// TIA Portal V15.1 export
// export: Created 2024-06-21T08:41:01.898082Z, ExportSetting WithDefaults, DisplayName Totally Integrated Automation Portal, DisplayVersion V15.1 Update 5, DisplayName TIA Portal Openness, DisplayVersion V15.1 Update 5, DisplayName SINAMICS Startdrive Advanced, DisplayVersion V15.1, DisplayName G130, G150, S120, S150, SINAMICS MV, S210, DisplayVersion V15.1, DisplayName G110M, G120, G120C, G120D, G120P, DisplayVersion V15.1, DisplayName STEP 7 Professional, DisplayVersion V15.1 Update 5, DisplayName STEP 7 Safety, DisplayVersion V15.1, DisplayName WinCC Professional, DisplayVersion V15.1 Update 5, DisplayName SIMATIC Visualization Architect, DisplayVersion V15.1
FUNCTION_BLOCK "LMovFnc2Pos"   // FB1102, FBD
TITLE = LMovFnc2Pos
{ S7_Optimized_Access := 'TRUE' }
AUTHOR : VCC
FAMILY : Tooling
VERSION : 0.1
// =============================================================================
// This module will be used for the steering of a two Position movement.
// It will get the commands from different Modes, evaluate the status of the 
// Interlock and give the command to the Actuator or direct to simple outputs.
// =============================================================================
// stored: AutoNumber false, IsIECCheckEnabled false, IsRetainMemResEnabled false, MemoryReserve 100, SetENOAutomatically False, UDAEnableTagReadback false
   VAR_INPUT
      I_PosSet { ExternalAccessible := 'False'; ExternalVisible := 'False'; ExternalWritable := 'False'} : Bool;   // Position Set detection or summary / Position Set Detection
      I_PosRes { ExternalAccessible := 'False'; ExternalVisible := 'False'; ExternalWritable := 'False'} : Bool;   // Position Reset detection or summary / Position Reset Detection
      I_PBSet { ExternalAccessible := 'False'; ExternalVisible := 'False'; ExternalWritable := 'False'} : Bool;   // Push button for Set direction (used in manual with button OP panels )
      I_PBReset { ExternalAccessible := 'False'; ExternalVisible := 'False'; ExternalWritable := 'False'} : Bool;   // Push button for reset direcion (used in manual with pushbutton OP panels) / Push button for Reset direction (used in manual with Pushbutton OP panels)
      I_SetBegin { ExternalAccessible := 'False'; ExternalVisible := 'False'; ExternalWritable := 'False'} : Bool;   // Function Set begin selection
      I_ResBegin { ExternalAccessible := 'False'; ExternalVisible := 'False'; ExternalWritable := 'False'} : Bool;   // Function Reset begin selection
      I_SetIntlkOK { ExternalAccessible := 'False'; ExternalVisible := 'False'; ExternalWritable := 'False'} : Bool;   // Set Interlock
      I_ResIntlkOK { ExternalAccessible := 'False'; ExternalVisible := 'False'; ExternalWritable := 'False'} : Bool;   // Reset Interlock
      I_SafetyOk { ExternalAccessible := 'False'; ExternalVisible := 'False'; ExternalWritable := 'False'} : Bool;   // Safety Ok
      I_HardwareOk { ExternalAccessible := 'False'; ExternalVisible := 'False'; ExternalWritable := 'False'} : Bool;   // Safety Ok / Hardware Ok
   END_VAR
   VAR_OUTPUT
      O_CmdSet { ExternalAccessible := 'False'; ExternalVisible := 'False'; ExternalWritable := 'False'} : Bool;   // Command to activate Set movement / Command to Activate Set movement
      O_CmdRes { ExternalAccessible := 'False'; ExternalVisible := 'False'; ExternalWritable := 'False'} : Bool;   // Command to activate Reset movement / Command to Activate Reset movement
      O_FuncRunning { ExternalAccessible := 'False'; ExternalVisible := 'False'; ExternalWritable := 'False'} : Bool;   // Signal that the function is running
      O_FuncBusyTM { ExternalAccessible := 'False'; ExternalVisible := 'False'; ExternalWritable := 'False'} : Bool;   // Memory Signal that the function is busy
      O_SetFinished { ExternalAccessible := 'False'; ExternalVisible := 'False'; ExternalWritable := 'False'} : Bool;   // Function Set finished to Master Sequencing
      O_ResFinished { ExternalAccessible := 'False'; ExternalVisible := 'False'; ExternalWritable := 'False'} : Bool;   // Function Reset finished to Master Sequencing
      O_IntlkSetAlm { ExternalAccessible := 'False'; ExternalVisible := 'False'; ExternalWritable := 'False'} : Bool;   // Alarm interlock Set / Alarm Interlock Set
      O_IntlkResAlm { ExternalAccessible := 'False'; ExternalVisible := 'False'; ExternalWritable := 'False'} : Bool;   // Alarm interlock Reset / Alarm Interlock Reset
      O_FuncIsSelInMan { ExternalAccessible := 'False'; ExternalVisible := 'False'; ExternalWritable := 'False'} : Bool;   // The function is selected in manual mode / The function is Selected in manual Mode
      O_LED { ExternalAccessible := 'False'; ExternalVisible := 'False'; ExternalWritable := 'False'} : Bool;   // LED-indication / LED - Indication
      O_AlarmABCondition { ExternalAccessible := 'False'; ExternalVisible := 'False'; ExternalWritable := 'False'} : Bool;   // Alarms AB condition / Alarm AB Condition
   END_VAR
   VAR_IN_OUT
      IO_Modes : "Modes";   // Modes
      H_HMI : "H_HMI";   // Animation
      H_MovFnc2Pos : "H_MovFnc2Pos";   // Animation
      H_FncSelInHMI { ExternalAccessible := 'False'; ExternalVisible := 'False'; ExternalWritable := 'False'} : Bool;   // This function is selected to run from HMI / This function is Selected to run from HMI
      C_AlarmResetUsed { ExternalAccessible := 'False'; ExternalVisible := 'False'; ExternalWritable := 'False'} : Bool;   // If true, the alrms will be stored untill reseted / If TRUE The Alarms will be stored untill Reseted
      C_EnableMemBegin { ExternalAccessible := 'False'; ExternalVisible := 'False'; ExternalWritable := 'False'} : Bool;   // Enable memory Begin (Command request is memorised until pos reached) / Enable memory Begin (Command Request is memorised until pos reached)
      C_EnIntlkAlm { ExternalAccessible := 'False'; ExternalVisible := 'False'; ExternalWritable := 'False'} : Bool := TRUE;   // Enable Interlock Alarm
      C_SetReset { ExternalAccessible := 'False'; ExternalVisible := 'False'; ExternalWritable := 'False'} : Bool;   // Enable Set Reset Functionality ( If enabled output is kept until the Cmd direction is changed )
      C_ManualClampCmdSet { ExternalAccessible := 'False'; ExternalVisible := 'False'; ExternalWritable := 'False'} : Bool;   // Manual Clamp Set
      C_ManualClampCmdRes { ExternalAccessible := 'False'; ExternalVisible := 'False'; ExternalWritable := 'False'} : Bool;   // Manual Clamp Reset
      C_ForceManual { ExternalAccessible := 'False'; ExternalVisible := 'False'; ExternalWritable := 'False'} : Bool := FALSE;   // Force Manual
   END_VAR
   VAR
      ResetAlarm { ExternalAccessible := 'False'; ExternalVisible := 'False'; ExternalWritable := 'False'} : Bool;   // Reset Alarm Memory
      CmdSetRequest { ExternalAccessible := 'False'; ExternalVisible := 'False'; ExternalWritable := 'False'} : Bool;   // Set Command request to activate the interlock / Set Command Request to Activate the Interlock
      CmdResRequest { ExternalAccessible := 'False'; ExternalVisible := 'False'; ExternalWritable := 'False'} : Bool;   // Reset Command request to activate the interlock / Reset Command Request to Activate the Interlock
      EdgeStopDetSet { ExternalAccessible := 'False'; ExternalVisible := 'False'; ExternalWritable := 'False'} : Bool;   // Edge on stop detection to be abble to go over it in force manual
      EdgeStopDetRes { ExternalAccessible := 'False'; ExternalVisible := 'False'; ExternalWritable := 'False'} : Bool;   // Edge on stop detection to be abble to go over it in force manual
      IntlkSetAlm { ExternalAccessible := 'False'; ExternalVisible := 'False'; ExternalWritable := 'False'} : Bool;   // Alarm interlock Set / Alarm Interlock Set
      IntlkResAlm { ExternalAccessible := 'False'; ExternalVisible := 'False'; ExternalWritable := 'False'} : Bool;   // Alarm interlock Reset / Alarm Interlock Reset
      CmdSet { ExternalAccessible := 'False'; ExternalVisible := 'False'; ExternalWritable := 'False'} : Bool;   // Command to activate Set movement / Command to Activate Set movement
      CmdRes { ExternalAccessible := 'False'; ExternalVisible := 'False'; ExternalWritable := 'False'} : Bool;   // Command to activate Reset movement / Command to Activate Reset movement
      IntlkSetAlmCond { ExternalAccessible := 'False'; ExternalVisible := 'False'; ExternalWritable := 'False'} : Bool;   // Alarm interlock Set condition / Alarm Interlock Set condition
      IntlkResAlmCond { ExternalAccessible := 'False'; ExternalVisible := 'False'; ExternalWritable := 'False'} : Bool;   // Alarm interlock Reset condition / Alarm Interlock Reset condition
      FuncRunning { ExternalAccessible := 'False'; ExternalVisible := 'False'; ExternalWritable := 'False'} : Bool;   // Function is running
      FuncBusyTM { ExternalAccessible := 'False'; ExternalVisible := 'False'; ExternalWritable := 'False'} : Bool;   // Memory Signal that the function is busy
      AlmFilterResult { ExternalAccessible := 'False'; ExternalVisible := 'False'; ExternalWritable := 'False'} : Bool;   // Alarm filter result
      _AlarmTimer { ExternalAccessible := 'False'; ExternalVisible := 'False'; ExternalWritable := 'False'} : "LTimer";
   END_VAR
   VAR_TEMP   // added for the SCL form of the ladder/FBD networks
      _w1 : Bool;
   END_VAR
BEGIN

REGION Network 1: **** 2.2 - Alarms - Alarm Generation **** Alarm Filter
   // Alarm Filter
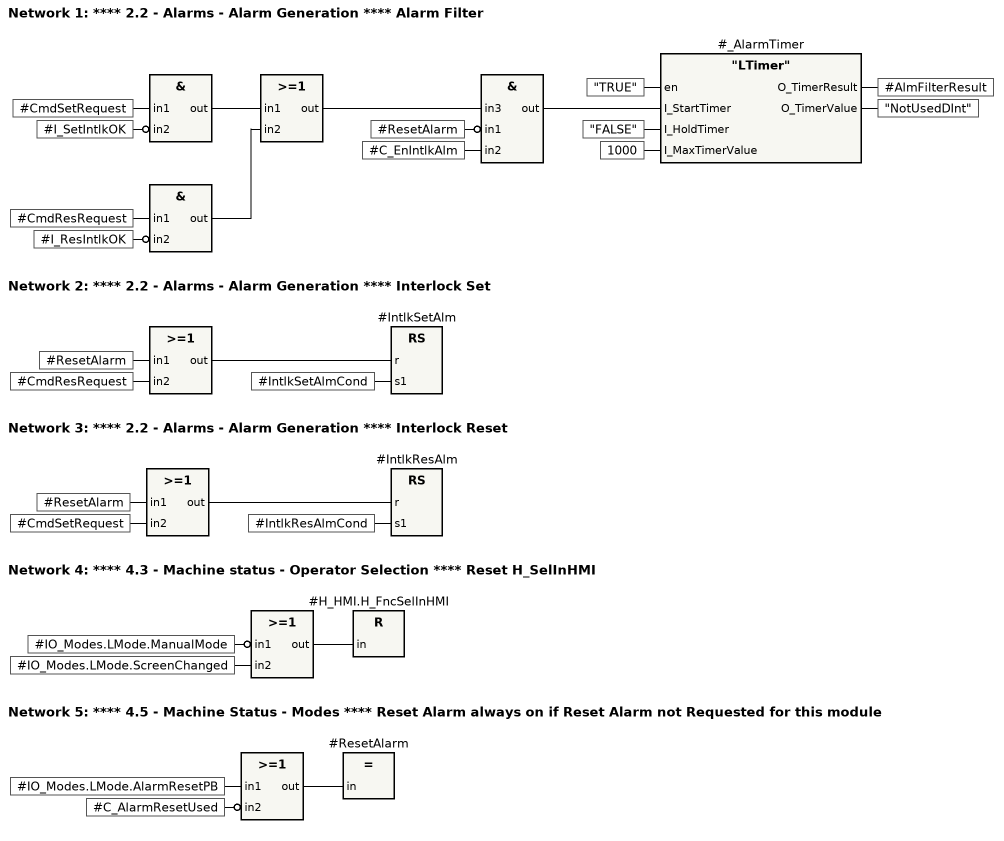
   IF "TRUE" THEN
       #_AlarmTimer(I_StartTimer := ((#CmdSetRequest AND NOT #I_SetIntlkOK) OR (#CmdResRequest AND NOT #I_ResIntlkOK)) AND NOT #ResetAlarm AND #C_EnIntlkAlm,   // "LTimer"
                    I_HoldTimer := "FALSE",
                    I_MaxTimerValue := 1000,
                    O_TimerResult => #AlmFilterResult,
                    O_TimerValue => "NotUsedDInt");
   END_IF;
END_REGION

REGION Network 2: **** 2.2 - Alarms - Alarm Generation **** Interlock Set
   // Interlock Set
   IF #ResetAlarm OR #CmdResRequest THEN
       #IntlkSetAlm := FALSE;   // RS flip-flop
   END_IF;
   IF #IntlkSetAlmCond THEN #IntlkSetAlm := TRUE; END_IF;
END_REGION

REGION Network 3: **** 2.2 - Alarms - Alarm Generation **** Interlock Reset
   // Interlock Reset
   IF #ResetAlarm OR #CmdSetRequest THEN
       #IntlkResAlm := FALSE;   // RS flip-flop
   END_IF;
   IF #IntlkResAlmCond THEN #IntlkResAlm := TRUE; END_IF;
END_REGION

REGION Network 4: **** 4.3 - Machine status - Operator Selection **** Reset H_SelInHMI
   // Reset H_SelInHMI
   IF NOT #IO_Modes.LMode.ManualMode OR #IO_Modes.LMode.ScreenChanged THEN
       #H_HMI.H_FncSelInHMI := FALSE;
   END_IF;
END_REGION

REGION Network 5: **** 4.5 - Machine Status - Modes **** Reset Alarm always on if Reset Alarm not Requested for this module
   // Reset Alarm always on if Reset Alarm not Requested for this module
   #ResetAlarm := #IO_Modes.LMode.AlarmResetPB OR NOT #C_AlarmResetUsed;
END_REGION

REGION Network 6: **** 4.6 - Machine Status - Indication **** Icon Animation
   // Icon Animation
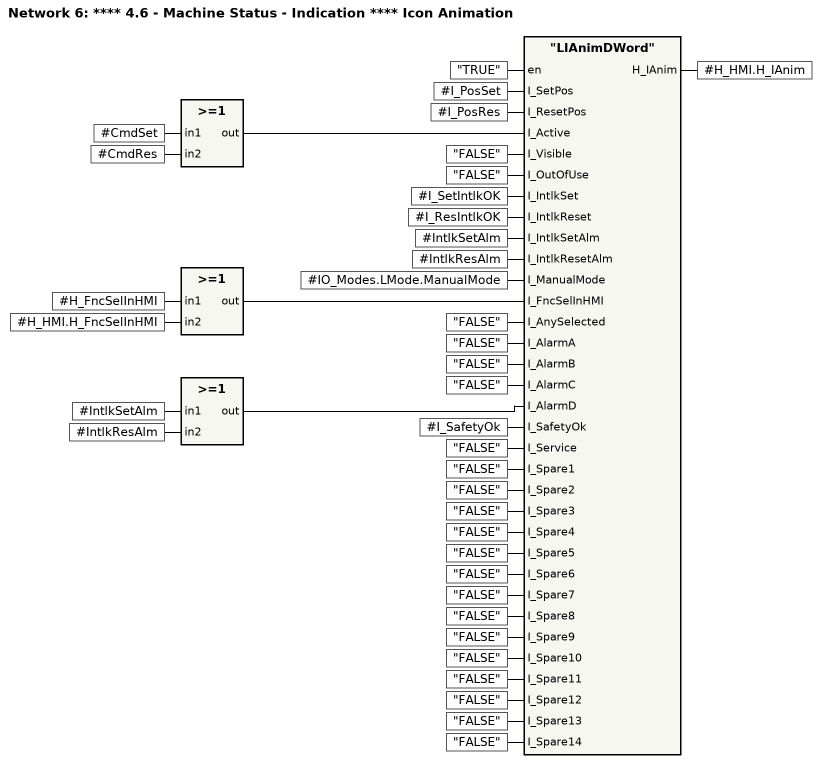
   IF "TRUE" THEN
       "LIAnimDWord"(I_SetPos := #I_PosSet,
                     I_ResetPos := #I_PosRes,
                     I_Active := #CmdSet OR #CmdRes,
                     I_Visible := "FALSE",
                     I_OutOfUse := "FALSE",
                     I_IntlkSet := #I_SetIntlkOK,
                     I_IntlkReset := #I_ResIntlkOK,
                     I_IntlkSetAlm := #IntlkSetAlm,
                     I_IntlkResetAlm := #IntlkResAlm,
                     I_ManualMode := #IO_Modes.LMode.ManualMode,
                     I_FncSelInHMI := #H_FncSelInHMI OR #H_HMI.H_FncSelInHMI,
                     I_AnySelected := "FALSE",
                     I_AlarmA := "FALSE",
                     I_AlarmB := "FALSE",
                     I_AlarmC := "FALSE",
                     I_AlarmD := #IntlkSetAlm OR #IntlkResAlm,
                     I_SafetyOk := #I_SafetyOk,
                     I_Service := "FALSE",
                     I_Spare1 := "FALSE",
                     I_Spare2 := "FALSE",
                     I_Spare3 := "FALSE",
                     I_Spare4 := "FALSE",
                     I_Spare5 := "FALSE",
                     I_Spare6 := "FALSE",
                     I_Spare7 := "FALSE",
                     I_Spare8 := "FALSE",
                     I_Spare9 := "FALSE",
                     I_Spare10 := "FALSE",
                     I_Spare11 := "FALSE",
                     I_Spare12 := "FALSE",
                     I_Spare13 := "FALSE",
                     I_Spare14 := "FALSE",
                     H_IAnim => #H_HMI.H_IAnim);
   END_IF;
END_REGION

REGION Network 7: **** 4.6 - Machine Status - Indication **** Animation
   // Animation
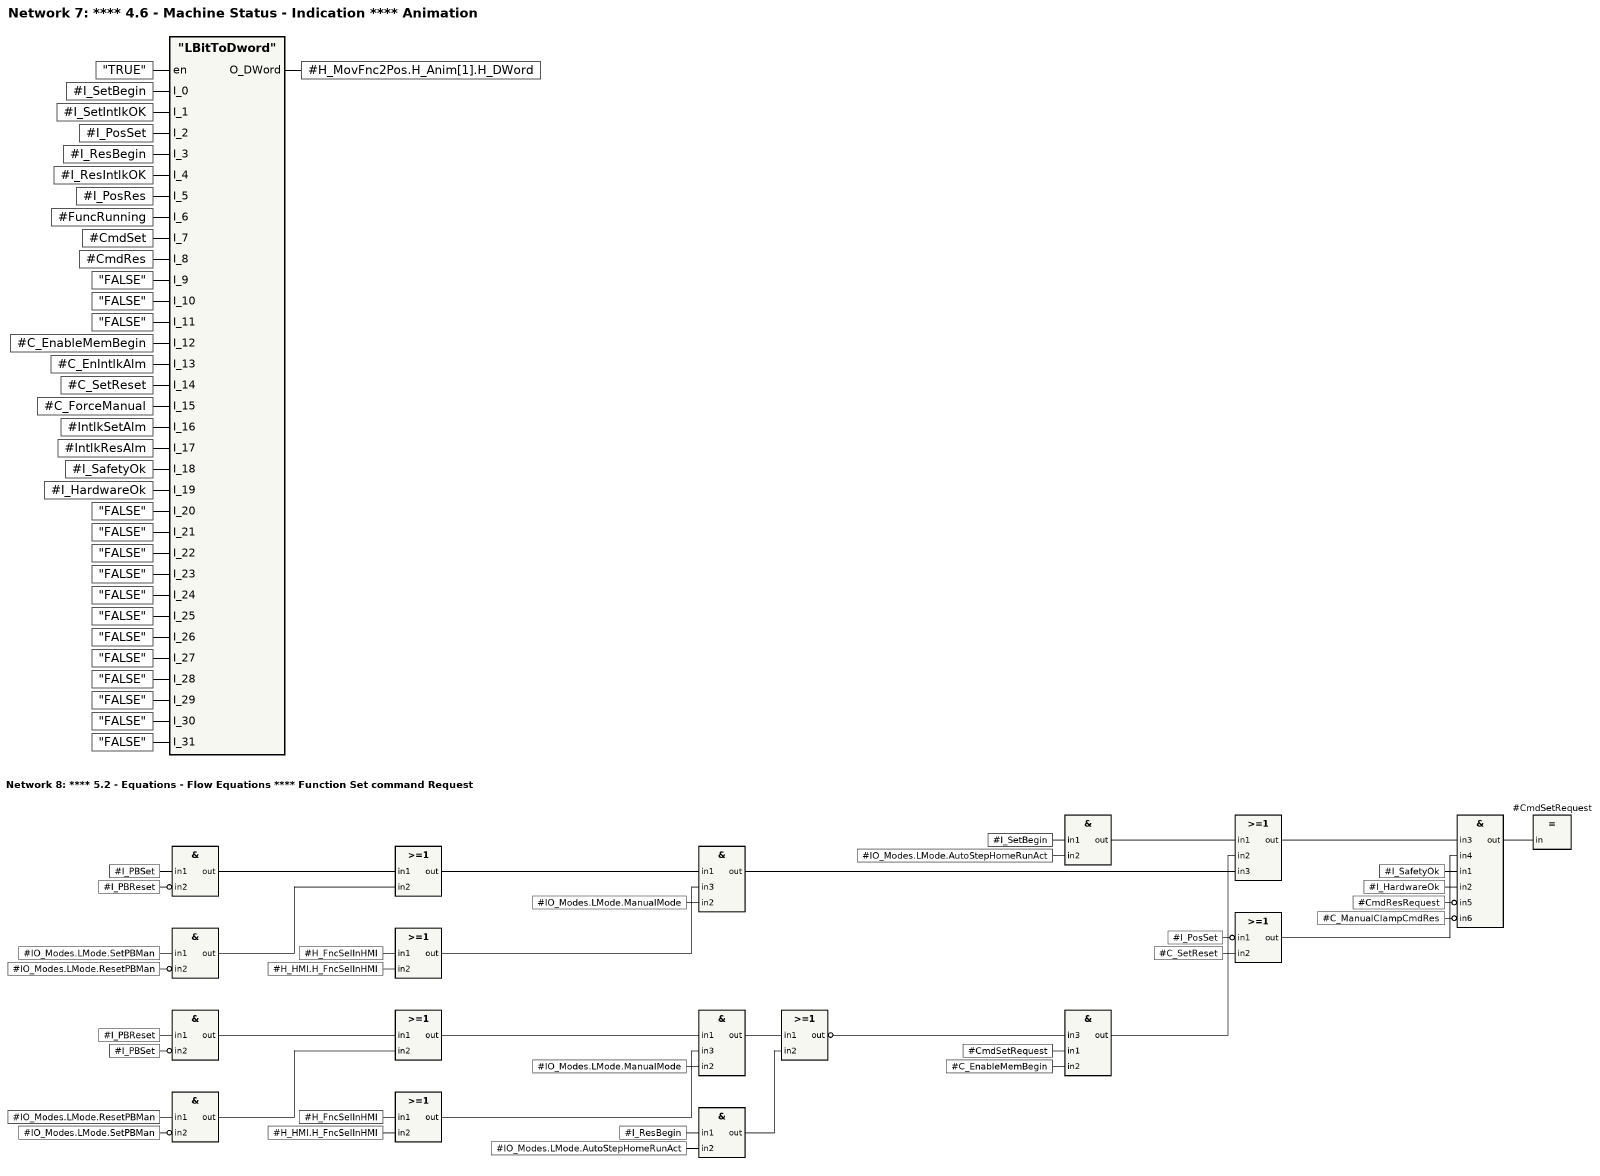
   IF "TRUE" THEN
       "LBitToDword"(I_0 := #I_SetBegin,
                     I_1 := #I_SetIntlkOK,
                     I_2 := #I_PosSet,
                     I_3 := #I_ResBegin,
                     I_4 := #I_ResIntlkOK,
                     I_5 := #I_PosRes,
                     I_6 := #FuncRunning,
                     I_7 := #CmdSet,
                     I_8 := #CmdRes,
                     I_9 := "FALSE",
                     I_10 := "FALSE",
                     I_11 := "FALSE",
                     I_12 := #C_EnableMemBegin,
                     I_13 := #C_EnIntlkAlm,
                     I_14 := #C_SetReset,
                     I_15 := #C_ForceManual,
                     I_16 := #IntlkSetAlm,
                     I_17 := #IntlkResAlm,
                     I_18 := #I_SafetyOk,
                     I_19 := #I_HardwareOk,
                     I_20 := "FALSE",
                     I_21 := "FALSE",
                     I_22 := "FALSE",
                     I_23 := "FALSE",
                     I_24 := "FALSE",
                     I_25 := "FALSE",
                     I_26 := "FALSE",
                     I_27 := "FALSE",
                     I_28 := "FALSE",
                     I_29 := "FALSE",
                     I_30 := "FALSE",
                     I_31 := "FALSE",
                     O_DWord => #H_MovFnc2Pos.H_Anim[1].H_DWord);
   END_IF;
END_REGION

REGION Network 8: **** 5.2 - Equations - Flow Equations **** Function Set command Request
   // Function Set command Request
   #CmdSetRequest := ((#I_SetBegin AND #IO_Modes.LMode.AutoStepHomeRunAct) OR (NOT ((((#I_PBReset AND NOT #I_PBSet) OR (#IO_Modes.LMode.ResetPBMan AND NOT #IO_Modes.LMode.SetPBMan)) AND (#H_FncSelInHMI OR #H_HMI.H_FncSelInHMI) AND #IO_Modes.LMode.ManualMode) OR (#I_ResBegin AND #IO_Modes.LMode.AutoStepHomeRunAct)) AND #CmdSetRequest AND #C_EnableMemBegin) OR (((#I_PBSet AND NOT #I_PBReset) OR (#IO_Modes.LMode.SetPBMan AND NOT #IO_Modes.LMode.ResetPBMan)) AND (#H_FncSelInHMI OR #H_HMI.H_FncSelInHMI) AND #IO_Modes.LMode.ManualMode)) AND (NOT #I_PosSet OR #C_SetReset) AND #I_SafetyOk AND #I_HardwareOk AND NOT #CmdResRequest AND NOT #C_ManualClampCmdRes;
END_REGION

REGION Network 9: **** 5.2 - Equations - Flow Equations **** Function Reset command Request
   // Function Reset command Request
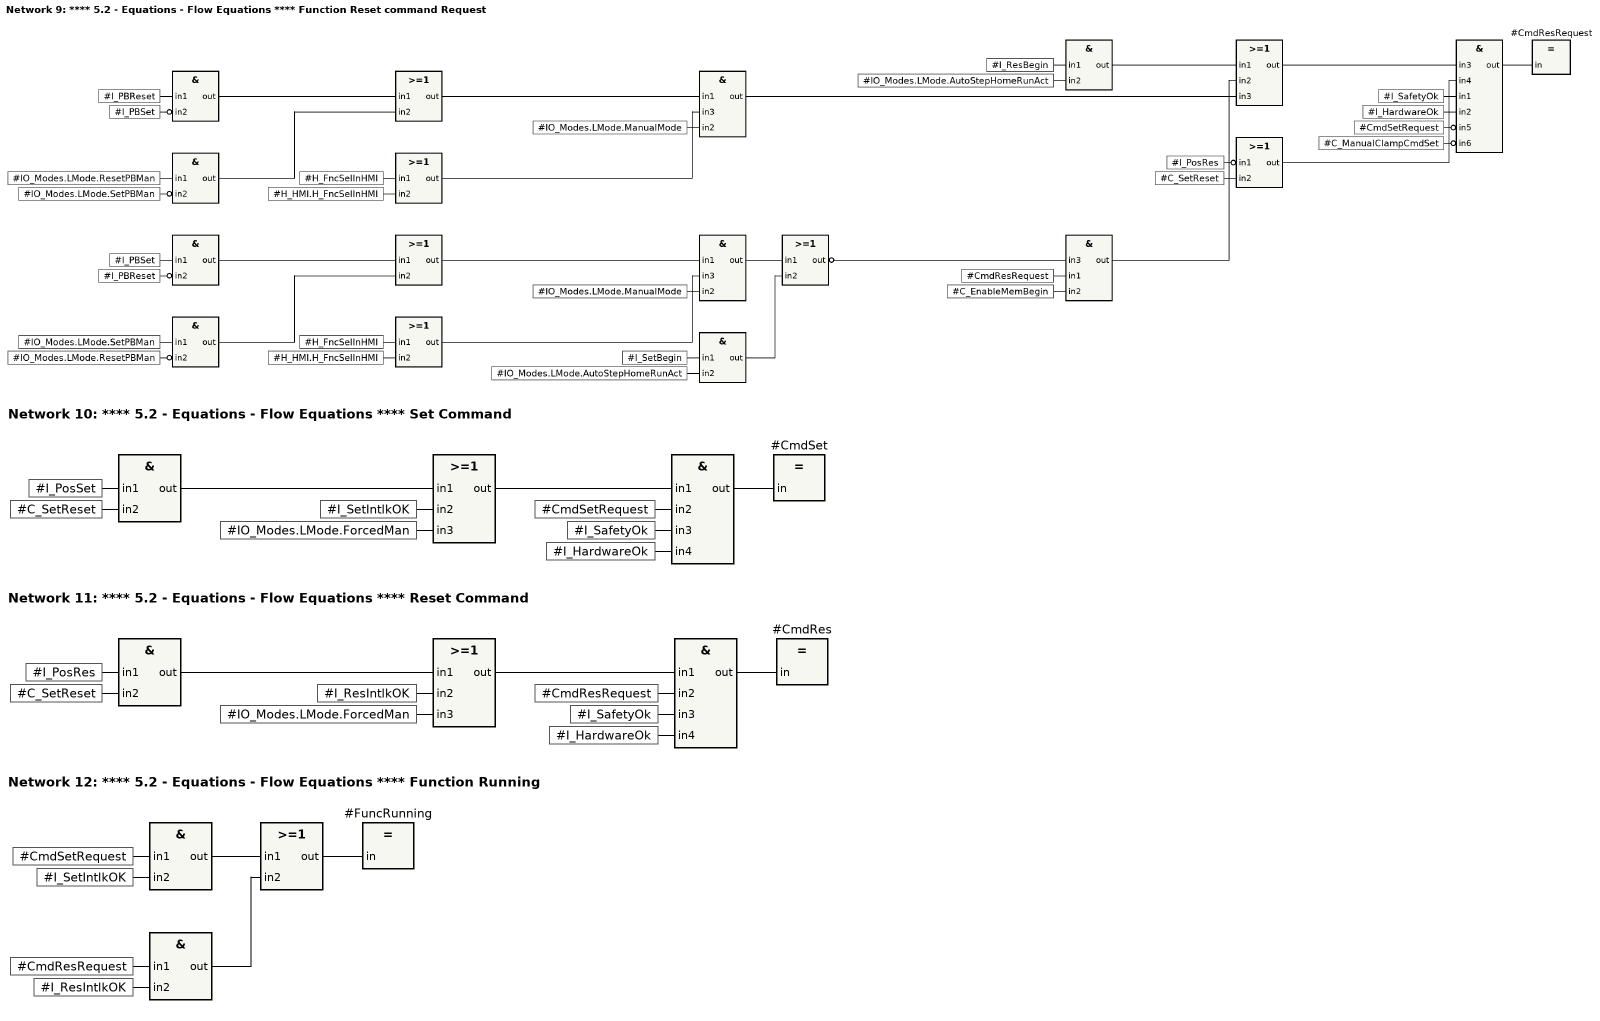
   #CmdResRequest := ((#I_ResBegin AND #IO_Modes.LMode.AutoStepHomeRunAct) OR (NOT ((((#I_PBSet AND NOT #I_PBReset) OR (#IO_Modes.LMode.SetPBMan AND NOT #IO_Modes.LMode.ResetPBMan)) AND (#H_FncSelInHMI OR #H_HMI.H_FncSelInHMI) AND #IO_Modes.LMode.ManualMode) OR (#I_SetBegin AND #IO_Modes.LMode.AutoStepHomeRunAct)) AND #CmdResRequest AND #C_EnableMemBegin) OR (((#I_PBReset AND NOT #I_PBSet) OR (#IO_Modes.LMode.ResetPBMan AND NOT #IO_Modes.LMode.SetPBMan)) AND (#H_FncSelInHMI OR #H_HMI.H_FncSelInHMI) AND #IO_Modes.LMode.ManualMode)) AND (NOT #I_PosRes OR #C_SetReset) AND #I_SafetyOk AND #I_HardwareOk AND NOT #CmdSetRequest AND NOT #C_ManualClampCmdSet;
END_REGION

REGION Network 10: **** 5.2 - Equations - Flow Equations **** Set Command
   // Set Command
   #CmdSet := ((#I_PosSet AND #C_SetReset) OR #I_SetIntlkOK OR #IO_Modes.LMode.ForcedMan) AND #CmdSetRequest AND #I_SafetyOk AND #I_HardwareOk;
END_REGION

REGION Network 11: **** 5.2 - Equations - Flow Equations **** Reset Command
   // Reset Command
   #CmdRes := ((#I_PosRes AND #C_SetReset) OR #I_ResIntlkOK OR #IO_Modes.LMode.ForcedMan) AND #CmdResRequest AND #I_SafetyOk AND #I_HardwareOk;
END_REGION

REGION Network 12: **** 5.2 - Equations - Flow Equations **** Function Running
   // Function Running
   #FuncRunning := (#CmdSetRequest AND #I_SetIntlkOK) OR (#CmdResRequest AND #I_ResIntlkOK);
END_REGION

REGION Network 13: **** 5.2 - Equations - Flow Equations **** Function Running Memory
   // Function Running Memory
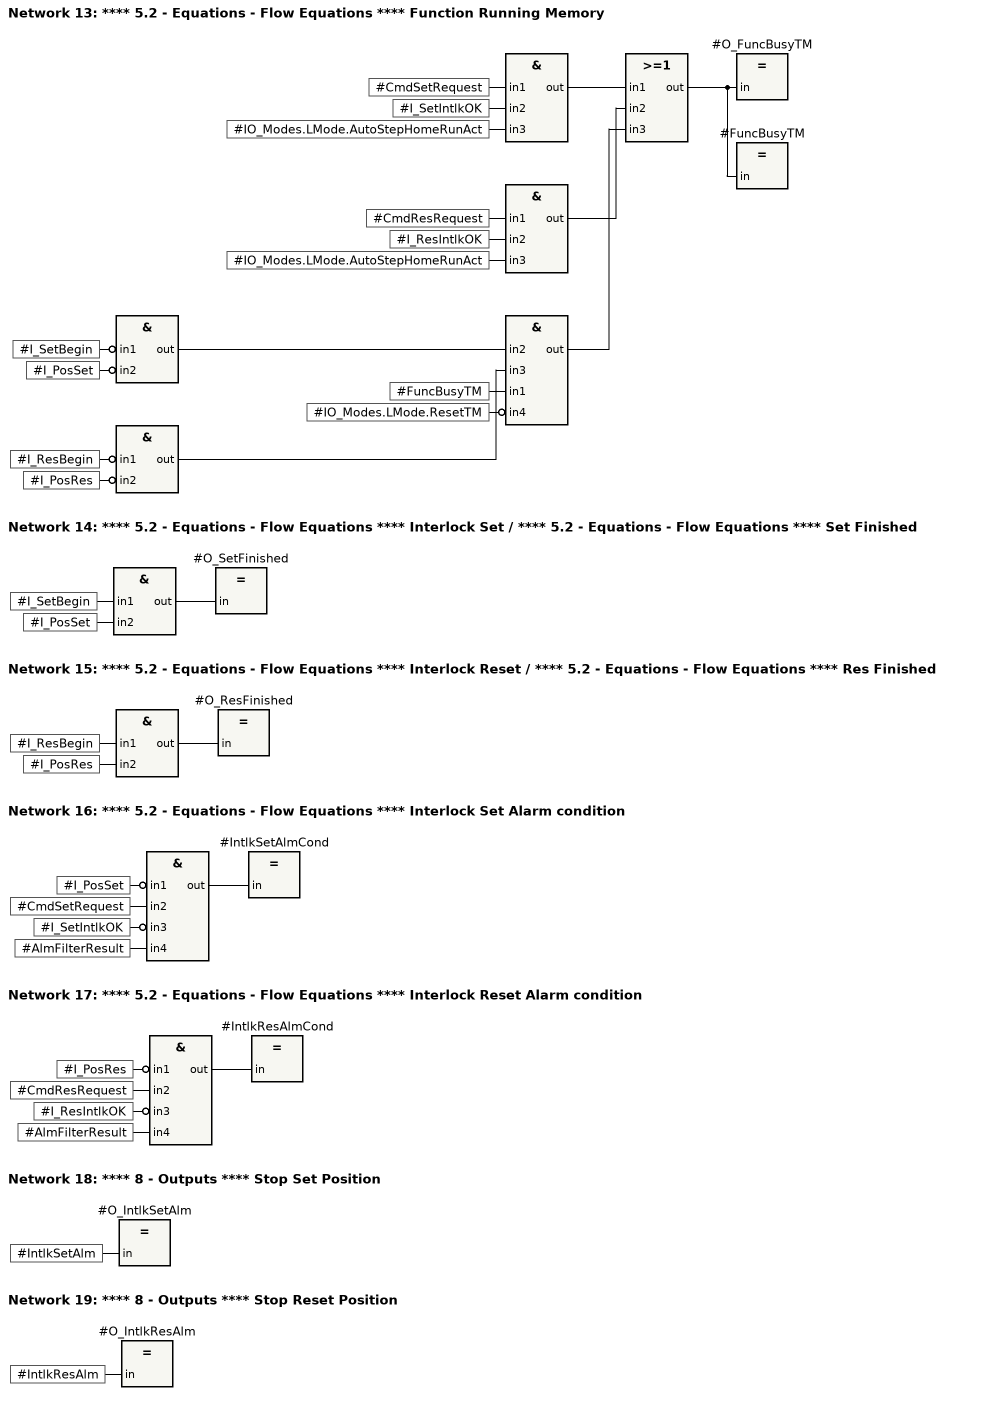
   #O_FuncBusyTM := (#CmdSetRequest AND #I_SetIntlkOK AND #IO_Modes.LMode.AutoStepHomeRunAct) OR (#CmdResRequest AND #I_ResIntlkOK AND #IO_Modes.LMode.AutoStepHomeRunAct) OR (NOT #I_SetBegin AND NOT #I_PosSet AND NOT #I_ResBegin AND NOT #I_PosRes AND #FuncBusyTM AND NOT #IO_Modes.LMode.ResetTM);
   #FuncBusyTM := #O_FuncBusyTM;
END_REGION

REGION Network 14: **** 5.2 - Equations - Flow Equations **** Interlock Set / **** 5.2 - Equations - Flow Equations **** Set Finished
   // Interlock Set
   #O_SetFinished := #I_SetBegin AND #I_PosSet;
END_REGION

REGION Network 15: **** 5.2 - Equations - Flow Equations **** Interlock Reset / **** 5.2 - Equations - Flow Equations **** Res Finished
   // Interlock Reset
   #O_ResFinished := #I_ResBegin AND #I_PosRes;
END_REGION

REGION Network 16: **** 5.2 - Equations - Flow Equations **** Interlock Set Alarm condition
   // Interlock Set Alarm condition
   #IntlkSetAlmCond := NOT #I_PosSet AND #CmdSetRequest AND NOT #I_SetIntlkOK AND #AlmFilterResult;
END_REGION

REGION Network 17: **** 5.2 - Equations - Flow Equations **** Interlock Reset Alarm condition
   // Interlock Reset Alarm condition
   #IntlkResAlmCond := NOT #I_PosRes AND #CmdResRequest AND NOT #I_ResIntlkOK AND #AlmFilterResult;
END_REGION

REGION Network 18: **** 8 - Outputs **** Stop Set Position
   // Stop Set Position
   #O_IntlkSetAlm := #IntlkSetAlm;
END_REGION

REGION Network 19: **** 8 - Outputs **** Stop Reset Position
   // Stop Reset Position
   #O_IntlkResAlm := #IntlkResAlm;
END_REGION

REGION Network 20: **** 8 - Outputs **** Function is Selected in manual Mode
   // Function is Selected in manual Mode
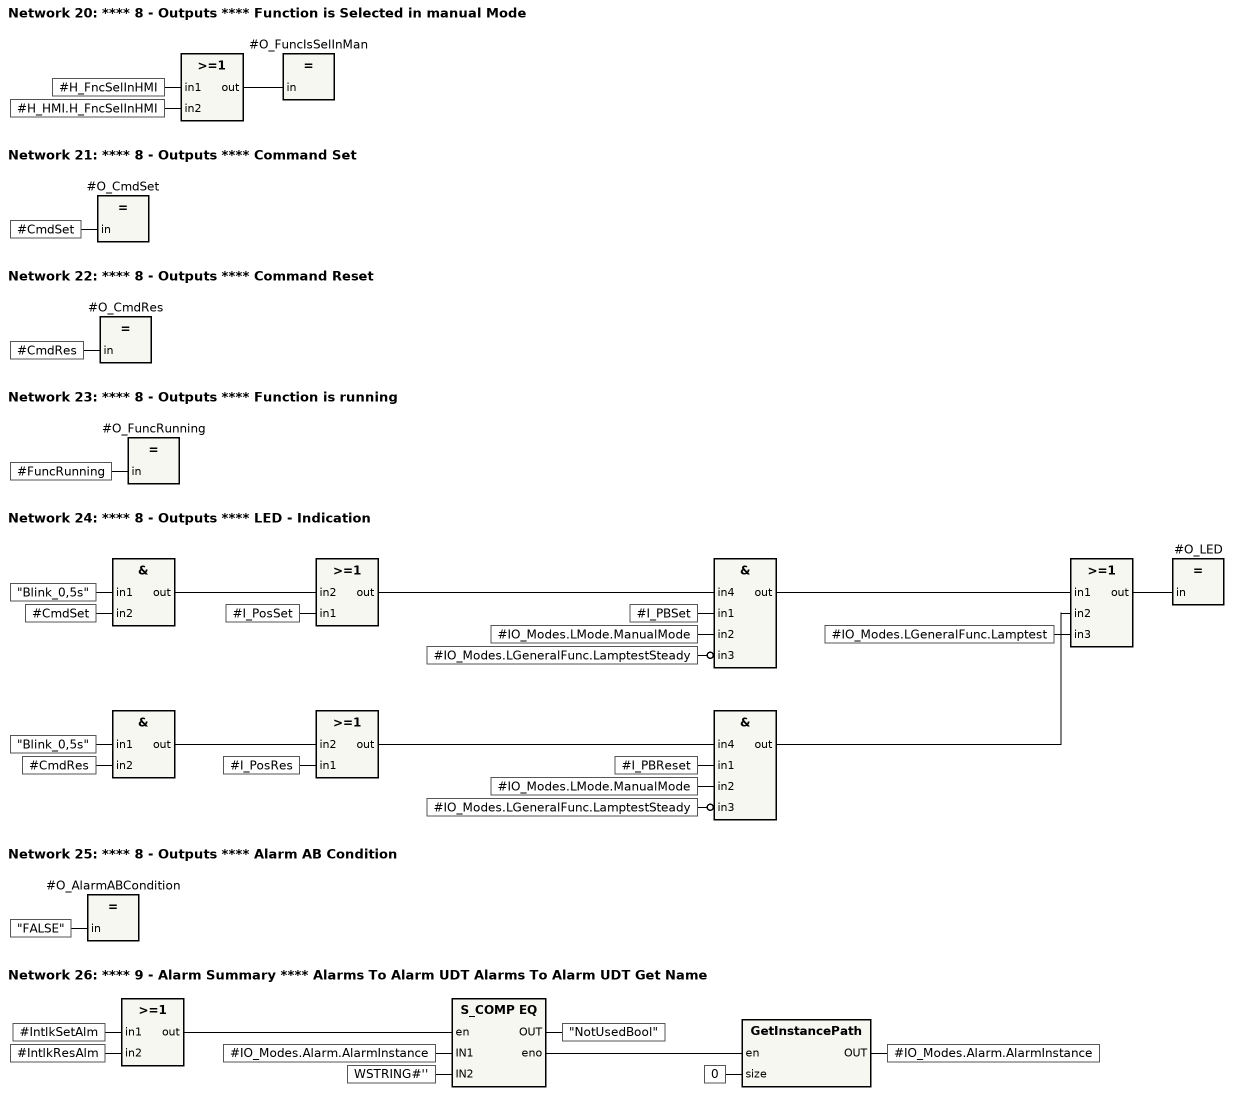
   #O_FuncIsSelInMan := #H_FncSelInHMI OR #H_HMI.H_FncSelInHMI;
END_REGION

REGION Network 21: **** 8 - Outputs **** Command Set
   // Command set
   #O_CmdSet := #CmdSet;
END_REGION

REGION Network 22: **** 8 - Outputs **** Command Reset
   // Command Reset
   #O_CmdRes := #CmdRes;
END_REGION

REGION Network 23: **** 8 - Outputs **** Function is running
   // Function is running
   #O_FuncRunning := #FuncRunning;
END_REGION

REGION Network 24: **** 8 - Outputs **** LED - Indication
   // LED - Indication
   #O_LED := ((("Blink_0,5s" AND #CmdSet) OR #I_PosSet) AND #I_PBSet AND #IO_Modes.LMode.ManualMode AND NOT #IO_Modes.LGeneralFunc.LamptestSteady) OR ((("Blink_0,5s" AND #CmdRes) OR #I_PosRes) AND #I_PBReset AND #IO_Modes.LMode.ManualMode AND NOT #IO_Modes.LGeneralFunc.LamptestSteady) OR #IO_Modes.LGeneralFunc.Lamptest;
END_REGION

REGION Network 25: **** 8 - Outputs **** Alarm AB Condition
   // Alarm AB Condition
   #O_AlarmABCondition := "FALSE";
END_REGION

REGION Network 26: **** 9 - Alarm Summary **** Alarms To Alarm UDT Alarms To Alarm UDT Get Name
   // Alarm / Alarm D
   S_COMP(EN := #IntlkSetAlm OR #IntlkResAlm,
          IN1 := #IO_Modes.Alarm.AlarmInstance,
          IN2 := WSTRING#'',
          OUT => "NotUsedBool",
          ENO => #_w1);
   IF #_w1 THEN GetInstancePath(size := 0, OUT => #IO_Modes.Alarm.AlarmInstance); END_IF;
END_REGION

REGION Network 27: **** 9 - Alarm Summary **** Alarms To Alarm UDT
   // Alarm / Alarm D
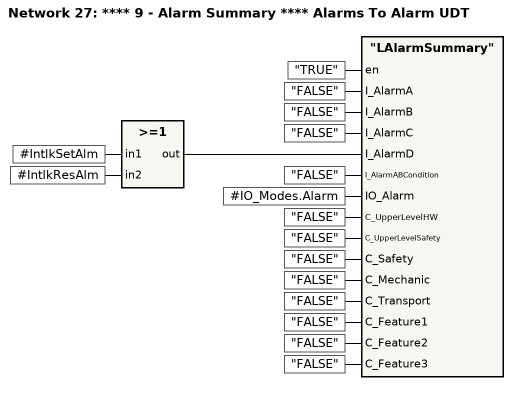
   IF "TRUE" THEN
       "LAlarmSummary"(I_AlarmA := "FALSE",
                       I_AlarmB := "FALSE",
                       I_AlarmC := "FALSE",
                       I_AlarmD := #IntlkSetAlm OR #IntlkResAlm,
                       I_AlarmABCondition := "FALSE",
                       IO_Alarm := #IO_Modes.Alarm,
                       C_UpperLevelHW := "FALSE",
                       C_UpperLevelSafety := "FALSE",
                       C_Safety := "FALSE",
                       C_Mechanic := "FALSE",
                       C_Transport := "FALSE",
                       C_Feature1 := "FALSE",
                       C_Feature2 := "FALSE",
                       C_Feature3 := "FALSE");
   END_IF;
END_REGION
END_FUNCTION_BLOCK
